// TIA Portal V21 export
FUNCTION "Cross-lock" : Void   // FC1, LAD
{ S7_Optimized_Access := 'TRUE' }
// stored: SetENOAutomatically false
   VAR_INPUT
      In1 : Bool;
      In2 : Bool;
   END_VAR
   VAR_OUTPUT
      Output1 : Bool;
      Output2 : Bool;
   END_VAR
BEGIN

REGION Network 1
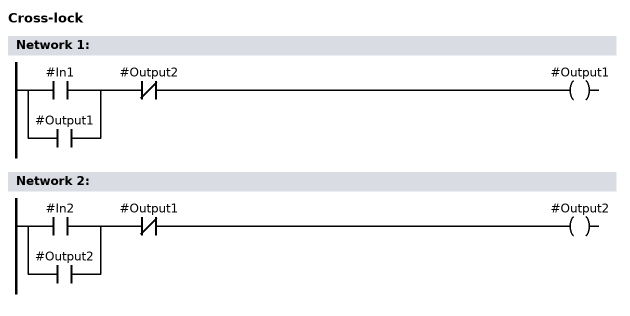
   RUNG wire#powerrail
      Contact( #In1 )
      wire#w1
      I_Contact( #Output2 )
      Coil( #Output1 )
   END_RUNG
   RUNG wire#powerrail
      Contact( #Output1 )
   END_RUNG wire#w1
   // the same network as SCL:
   #Output1 := (#In1 OR #Output1) AND NOT #Output2;
END_REGION

REGION Network 2
   RUNG wire#powerrail
      Contact( #In2 )
      wire#w1
      I_Contact( #Output1 )
      Coil( #Output2 )
   END_RUNG
   RUNG wire#powerrail
      Contact( #Output2 )
   END_RUNG wire#w1
   // the same network as SCL:
   #Output2 := (#In2 OR #Output2) AND NOT #Output1;
END_REGION
END_FUNCTION
